(* IEC 61131-3 sources: Lasal/CPU_5344_V01/Class/StringDll, 1 file *)

(* ---- StringDll.st ---- *)
(*!
<Class
	Name               = "StringDll"
	Revision           = "0.0"
	RealtimeTask       = "false"
	CyclicTask         = "false"
	BackgroundTask     = "false"
	Sigmatek           = "false"
	OSInterface        = "false"
	HighPriority       = "false"
	Automatic          = "false"
	UpdateMode         = "Prescan"
	SharedCommandTable = "true"
	Objectsize         = "(284,120)">
	<Channels>
		<Server Name="Handle" Visualized="false" Initialize="false" WriteProtected="false" Retentive="false"/>
	</Channels>
	<Network Name="StringDll">
		<!-- List of Components in this network -->
		<Components>
			<Object
				Name       = "_base"
				Class      = "String"
				Position   = "(218,120)"
				Visualized = "false">
				<Channels>
					<Server Name="Data"/>
					<Client Name="SingleRealloc" Value="1"/>
				</Channels>
			</Object>
		</Components>
		<Comments>
		</Comments>
		<!-- List of Connections in this network -->
		<Connections>
			<Connection Source="this.Data" Destination="_base.Data" Vertices="(1156,210),(984,210),"/>
		</Connections>
		<!-- Headerfiles -->
		<Options>
		</Options>
	</Network>
</Class>
*)
#pragma using String

StringDll : CLASS
: String
  //Servers:
	Handle 	: SvrCh_DINT;
  //Clients:
  //Variables:
		strTemp : ARRAY [0..255] OF DINT;

  //Functions:

	FUNCTION VIRTUAL GLOBAL Handle::Read
		VAR_OUTPUT
			output (EAX) 	: DINT;
		END_VAR;

	FUNCTION VIRTUAL GLOBAL Handle::Write
		VAR_INPUT
			input (EAX) 	: DINT;
		END_VAR
		VAR_OUTPUT
			result (EAX) 	: DINT;
		END_VAR;
  //Tables:
	FUNCTION @STD
		VAR_OUTPUT
			ret_code	: CONFSTATES;
		END_VAR;
	FUNCTION GLOBAL TAB @CT_;
END_CLASS;

FUNCTION VIRTUAL GLOBAL StringDll::Handle::Read
	VAR_OUTPUT
		output (EAX) 	: DINT;
	END_VAR

  Handle := (#strTemp[0])$dint;
	output := Handle;

END_FUNCTION

FUNCTION VIRTUAL GLOBAL StringDll::Handle::Write
	VAR_INPUT
		input (EAX) 	: DINT;
	END_VAR
	VAR_OUTPUT
		result (EAX) 	: DINT;
	END_VAR

	Handle := input;
  WriteDataOff(udLen:=255, udOff:=0, pData:=#strTemp[0]$usint);
 	result := Handle;

END_FUNCTION
